INTERFACE I_AssertMessageFormatter

METHOD LogAssertFailure
VAR_INPUT
    Expected : T_MaxString;
    Actual : T_MaxString;
    Message : T_MaxString;
    TestInstancePath : T_MaxString;
END_VAR
END_METHOD

END_INTERFACE

(* stored: Version 1.1.0.1
   Itf I_AssertMessageFormatter: Id {71246e7e-3534-44b1-a788-c1f37427a096}
   Method LogAssertFailure: Id {35efab01-6ac8-46a5-a5e1-adb4f1f5f9b2} *)
